Fanuc KAREL source: compact_preamble.KL

PROGRAM KT00943
%NOLOCKGROUP
VAR
ENTRY:INTEGER;PNAME : STRING[80];VNAME : STRING[80];STATUS:INTEGER;VALUE : VECTOR
BEGIN
ENTRY=0
PNAME=''
VNAME='VALUE'
GET_VAR(ENTRY,PNAME,VNAME,VALUE,STATUS)
END KT00943
